PROGRAM MAIN
VAR
END_VAR

END_PROGRAM

(* stored: Version 1.1.0.1, ProductVersion 3.1.4024.12
   POU MAIN: Id {840f8603-509d-05bb-33a9-60c87889393c}, SpecialFunc None *)
